PROGRAM MAIN
VAR
END_VAR

END_PROGRAM

(* stored: Version 1.1.0.1
   POU MAIN: Id {00d7d17e-f738-44c0-be49-dce4eda92388} *)
